FUNCTION_BLOCK CStringBuilderExample
VAR_INPUT
END_VAR
VAR_OUTPUT
END_VAR
VAR
	//run tests
	startClassAndInitializationTest, startSimpleUseTest : BOOL;

	
	simpleUseOutput1, simpleUseOutput2 : STRING(1000);

	
	StringBuilder : CStringBuilder; 
	Value : STRING(255) := 'Dieser Text ist genau 250 Zeichen lang und wird verwendet, um zu zeigen, wie TwinCAT 3 Strings handhabt. Es handelt sich um einen langen Satz, der viele verschiedene Themen behandelt, wie z.B. Programmierung, Automatisierungstechnik, SPS-Programmieru';
	currentString:  STRING(3000);
	pResult : POINTER TO BYTE;
	Stage, SimpleUseStage : INT;
	
	stStringBuilderPara : ST_StringBuilderPara := (MaxBufferSize:=3000);
	
 	boolExample : BOOL := TRUE;
    byteExample : BYTE := 16#FF;
    wordExample : WORD := 16#FFFF;
    dwordExample : DWORD := 16#FFFFFFFF;
    lwordExample : LWORD := 16#FFFFFFFFFFFFFFFF;
    sintExample : SINT := -128;
    intExample : INT := -32768;
    dintExample : DINT := -2147483648;
    lintExample : LINT := -9223372036854775808;
    usintExample : USINT := 255;
    uintExample : UINT := 65535;
    udintExample : UDINT := 4294967295;
    ulintExample : ULINT := 18446744073709551615;
    realExample : REAL := 1.0;
    lrealExample : LREAL := 1.0;
    timeExample : TIME := T#5s;
    dateExample : DATE := D#2023-01-01;
    todExample : TOD := TOD#12:00:00;
    dtExample : DT := DT#2023-01-01-12:00:00;
    stringExample : STRING := 'I am a string';
END_VAR

METHOD ClassAndInitialization : BOOL
VAR_INPUT
END_VAR
CASE Stage OF
	
	0:
		IF startClassAndInitializationTest THEN
			startClassAndInitializationTest := FALSE;
			StringBuilder.Init(pPara:=ADR(THIS^.stStringBuilderPara));
			Stage := 1;
		END_IF
		
	1:
		StringBuilder
            .Append(Value:='This is a bool: ')
            .AppendAny(Value:=boolExample)
            .Append(Value:=', This is a byte: ')
            .AppendAny(Value:=byteExample)
            .Append(Value:=', This is a word: ')
            .AppendAny(Value:=wordExample)
            .Append(Value:=', This is a dword: ')
            .AppendAny(Value:=dwordExample)
            .Append(Value:=', This is a lword: ')
            .AppendAny(Value:=lwordExample)
            .Append(Value:=', This is a sint: ')
            .AppendAny(Value:=sintExample)
            .Append(Value:=', This is an int: ')
            .AppendAny(Value:=intExample);
			
			//separation done, compiling + logging in needs pretty long for chains longer than 14
			StringBuilder
			.Append(Value:=', This is a dint: ')
            .AppendAny(Value:=dintExample)
            .Append(Value:=', This is a lint: ')
            .AppendAny(Value:=lintExample)
            .Append(Value:=', This is a usint: ')
            .AppendAny(Value:=usintExample)
            .Append(Value:=', This is a uint: ')
            .AppendAny(Value:=uintExample)
            .Append(Value:=', This is a udint: ')
            .AppendAny(Value:=udintExample)
            .Append(Value:=', This is a ulint: ')
            .AppendAny(Value:=ulintExample)
            .Append(Value:=', This is a real: ')
            .AppendAny(Value:=realExample);
			
			StringBuilder
            .Append(Value:=', This is an lreal: ')
            .AppendAny(Value:=lrealExample)
            .Append(Value:=', This is a time: ')
            .AppendAny(Value:=timeExample)
            .Append(Value:=', This is a date: ')
            .AppendAny(Value:=dateExample)
            .Append(Value:=', This is a tod: ')
            .AppendAny(Value:=todExample)
            .Append(Value:=', This is a dt: ')
            .AppendAny(Value:=dtExample)
            .Append(Value:=', This is a string: ')
            .AppendAny(Value:=stringExample);
			
			// add string in json format
			StringBuilder.Append('{"type":"')
			.Append('Name')
			.Append('","namespace":"')
			.Append('NameSpace1')
			.Append('","id":')
			.Append('10')
			.Append(',"count":')
			.Append('22')
			.Append(',"guid":"')
			.Append('7777-7777-7777-7777')
			.Append('"}');
		// show string data
		StringBuilder.Copy(pDest:=ADR(currentString), n:=SIZEOF(currentString));
		Stage := 2;
		
		2:
			StringBuilder.Clear();
			Stage := 0;
		
		
END_CASE
END_METHOD

METHOD SimpleUse : BOOL
VAR_INPUT
END_VAR
// build string, copy to destination

CASE SimpleUseStage OF


	0:
		IF THIS^.startSimpleUseTest THEN
			startSimpleUseTest := FALSE;
			//build string, copy to given destination
			BuildString(nSizeDest:=SIZEOF(simpleUseOutput1))
			.AppendAny(boolExample)
			.AppendAny(dintExample)
			.Copy(pDest:=ADR(simpleUseOutput1), n:=SIZEOF(simpleUseOutput1));
			SimpleUseStage := 1;
		END_IF
		
	1: //clear buffer, fill + copy to next string
		BuildString(nSizeDest:=SIZEOF(simpleUseOutput2))
		.Clear()
		.AppendAny(dwordExample)
		.AppendAny(dtExample)
		.AppendAny(stringExample)
		.Copy(pDest:=ADR(simpleUseOutput2), n:=SIZEOF(simpleUseOutput2));
		SimpleUseStage := 0;
	
	
	
	
END_CASE
END_METHOD

END_FUNCTION_BLOCK

(* stored: Version 1.1.0.1, ProductVersion 3.1.4024.13
   POU CStringBuilderExample: Id {447b65b5-cd1a-4395-a4b5-8fe33216f0df}, SpecialFunc None
   Method ClassAndInitialization: Id {9ca5d71e-b86e-4038-966d-0f5f3c1e1bc0}
   Method SimpleUse: Id {f437f28c-d69e-49c0-8953-8b8986bbba39} *)
